(* IEC 61131-3 sources: standardizer-tutorial-lib/src/Axis, 2 files *)

(* ---- ISpeedAxis.st ---- *)
NAMESPACE Simatic.Ax.Axis
    INTERFACE ISpeedAxis

        METHOD  Halt
        END_METHOD

        METHOD MoveVelocity
            VAR_INPUT
                Speed : LREAL;
                Direction : Direction;
            END_VAR
        END_METHOD

    END_INTERFACE

    TYPE
        Direction :
        (
            FORWARD,
            REVERSE
        );
    END_TYPE

END_NAMESPACE

(* ---- AnalogMotor.st ---- *)
USING Simatic.Ax.IO.Output;
NAMESPACE Simatic.Ax.Axis
    CLASS AnalogMotor IMPLEMENTS ISpeedAxis

        VAR PUBLIC
            qMotorSpeed : LRealOutput;
        END_VAR

        METHOD PUBLIC Halt
            qMotorSpeed.SetValue(0.0);
        END_METHOD

        METHOD PUBLIC MoveVelocity
            VAR_INPUT
                Speed : LREAL;
                Direction : Direction;
            END_VAR
            IF Direction = Direction#FORWARD THEN
                qMotorSpeed.SetValue(Speed);
            ELSE
                qMotorSpeed.SetValue(-1.0 * Speed);
            END_IF;

        END_METHOD
    END_CLASS

END_NAMESPACE
